// TIA Portal V16 export
// export: Created 2021-11-12T13:33:59.57236Z, ExportSetting WithDefaults, DisplayName Totally Integrated Automation Portal, DisplayVersion V16 Update 3, DisplayName TIA Portal Version Control Interface, DisplayVersion V16 Update 2, DisplayName TIA Portal Openness, DisplayVersion V16 Update 3, DisplayName SINAMICS Startdrive Advanced, DisplayVersion V16 Update 5, DisplayName SINAMICS Startdrive G130, G150, S120, S150, SINAMICS MV, S210, DisplayVersion V16 Update 5, DisplayName SINAMICS Startdrive G110M, G120, G120C, G120D, G120P, G115D, DisplayVersion V16 Update 5, DisplayName STEP 7 Professional, DisplayVersion V16 Update 3, DisplayName STEP 7 Safety, DisplayVersion V16, DisplayName WinCC UA Professional, DisplayVersion V16 Update 3
TYPE "UDT_COMM_BSN1_CRS"
// stored: IsFailsafeCompliant false
   STRUCT
      LiveBit : Bool;   // Periodical signal 5 Hz
      NoErr : Bool;   // No summary fault on the machine
      Aut : Bool;   // Machine is ready for automatic production
      AutRun : Bool;   // Machine is in mode for remote control (ICE) - automatic production
      Man : Bool;   // Machine is in manual mode
      Res_0_5 : Bool;
      Heating : Bool;   // Machine is in state heating
      Res_0_7 : Bool;
      Res_1_0 : Bool;
      Res_1_1 : Bool;
      Res_1_2 : Bool;
      Res_1_3 : Bool;
      Res_1_4 : Bool;
      Res_1_5 : Bool;
      Res_1_6 : Bool;
      Res_1_7 : Bool;
      Eject1Up : Bool;   // BSN1 - ejector 1 upper position
      Eject2Up : Bool;   // BSN1 - ejector 2 upper position
      Eject3Up : Bool;   // BSN1 - ejector 3 upper position
      Eject4Up : Bool;   // BSN1 - ejector 4 upper position
      Eject5Up : Bool;   // BSN1 - ejector 5 upper position
      Door2Up : Bool;   // Door 2 (left) opened
      Door1Up : Bool;   // Door 1 (right) opened
      Res_2_7 : Bool;
      Res_3_0 : Bool;
      Res_3_1 : Bool;
      Res_3_2 : Bool;
      Res_3_3 : Bool;
      Res_3_4 : Bool;
      Res_3_5 : Bool;
      Res_3_6 : Bool;
      Res_3_7 : Bool;
      Res_4_0 : Bool;
      Res_4_1 : Bool;
      Res_4_2 : Bool;
      Res_4_3 : Bool;
      Res_4_4 : Bool;
      Res_4_5 : Bool;
      Res_4_6 : Bool;
      Res_4_7 : Bool;
      Tact : Bool;   // belt is moving
      TactDone : Bool;   // belt reached destination position
      PartOnOut : Bool;   // part in output row - BG50.3
      PartBehDoor : Bool;   // part behind the doors - BG52.4
      Res_5_6 : Bool;
      Res_5_7 : Bool;
      Res_5_8 : Bool;
      Res_5_9 : Bool;
      Res_6_0 : Bool;
      Res_6_1 : Bool;
      Res_6_2 : Bool;
      Res_6_3 : Bool;
      Res_6_4 : Bool;
      Res_6_5 : Bool;
      Res_6_6 : Bool;
      Res_6_7 : Bool;
      Res_7_0 : Bool;
      Res_7_1 : Bool;
      Res_7_2 : Bool;
      Res_7_3 : Bool;
      Res_7_4 : Bool;
      Res_7_5 : Bool;
      Res_7_6 : Bool;
      Res_7_7 : Bool;
      Res_8_0 : Bool;
      Res_8_1 : Bool;
      Res_8_2 : Bool;
      Res_8_3 : Bool;
      Res_8_4 : Bool;
      Res_8_5 : Bool;
      Res_8_6 : Bool;
      Res_8_7 : Bool;
      Res_9_0 : Bool;
      Res_9_1 : Bool;
      Res_9_2 : Bool;
      Res_9_3 : Bool;
      Res_9_4 : Bool;
      Res_9_5 : Bool;
      Res_9_6 : Bool;
      Res_9_7 : Bool;
      ActTempSetpointZ1 : Int;   // actual temperature setpoint in zone 1 [°C]
      ActTempZ1 : Int;   // actual temperature in zone 1 [°C]
      ActTempSetpointZ2 : Int;   // actual temperature setpoint in zone 2 [°C]
      ActTempZ2 : Int;   // actual temperature in zone 2 [°C]
      ActTempSetpointZ3 : Int;   // actual temperature setpoint in zone 3 [°C]
      ActTempZ3 : Int;   // actual temperature in zone 3 [°C]
      ActTempSetpointZ4 : Int;   // actual temperature setpoint in zone 4 [°C]
      ActTempZ4 : Int;   // actual temperature in zone 4 [°C]
      ActTempSetpointZ5 : Int;   // actual temperature setpoint in zone 5 [°C]
      ActTempZ5 : Int;   // actual temperature in zone 5 [°C]
      ActTactTimeSetpoint : Int := 0;   // actual setpoint tact time [s]
      ActStepLengthSetpoint : Int := 0;   // actual setpoint step length
      ActBeltExtens : Int;   // actual belt extension [mm]
      ActBurnerHigh : Int;   // actual setpoint burner high [mm]
      Res_I38 : Int;
      Res_I40 : Int;
      Res_I42 : Int;
      Res_I44 : Int;
      Res_I46 : Int;
      Res_I48 : Int;
      Res_I50 : Int;
      Res_I52 : Int;
      Res_I54 : Int;
      Res_I56 : Int;
      Res_I58 : Int;
      Res_I60 : Int;
      Res_I62 : Int;
   END_STRUCT;
END_TYPE
